{attribute clr[Container(Layout.Stack)]}
{attribute clr[Group(Layout.GroupBox)]}
{attribute addProperty PreviousPort "Unknown"}
TYPE EtcSlaveBoxBase_77A0E4A7 EXTENDS EtcSlaveBase_82538BE2 :
STRUCT
END_STRUCT
END_TYPE

(* stored: Version 1.2.0.0
   DUT EtcSlaveBoxBase_77A0E4A7: Id {aeea0591-190f-4a02-b4f7-ac0152452496} *)
